(* CoDeSys 2.3 export: LOWPASS_INIT.EXP *)

(* POU 05_Basic_Calc/Lowpass_init, ST *)
FUNCTION_BLOCK Lowpass_init
VAR_INPUT
	tTime_constant: TIME;
	iCycle_time: INT;
END_VAR
VAR_OUTPUT
END_VAR
VAR_IN_OUT
	iDivisor: INT;
END_VAR

VAR
	iTime_constant:INT;
END_VAR
iTime_constant:=TIME_TO_INT(tTime_constant);

iCycle_time := MAX(1,iCycle_time );	(*not zero*)
iTime_constant := LIMIT(iCycle_time, iTime_constant, iTime_constant); (*Time constant min. Cycle_time*)

iDivisor:=iTime_constant / iCycle_time;
END_FUNCTION_BLOCK
